{attribute 'qualified_only'}
{attribute 'strict'}
TYPE E_SpeedModeBackendController_EMS :
(
	eSlow			:= 0,
	eBalanced 		:= 1,
	eFast			:= 2
);
END_TYPE

(* stored: Version 1.1.0.1, ProductVersion 3.1.4024.9
   DUT E_SpeedModeBackendController_EMS: Id {453f0a7a-605a-4baf-aab2-a7dfc2c64dfe} *)
